(* CODESYS project SPT_Drives.library
   Company: Beckhoff Automation LLC
   DefaultNamespace: SPT_Drives
   Version: 3.0.2
   Placeholder: SPT Drives
   Title: SPT Drives

Project tree, tasks and I/O mapping:
  libraries: SPT Base Types, * (Beckhoff Automation LLC); SPT NC Axis, * (Beckhoff Automation LLC); Tc2_MC2, * (Beckhoff Automation GmbH); Tc2_NcDrive, * (Beckhoff Automation GmbH); Tc3_Module, * (Beckhoff Automation GmbH)
  Beckhoff/
    AX5000/
      function block FB_ResetRoutine_SoEDrive [ST]: Axis, CyclicLogic, Execute
    AX8000/
      function block FB_ResetRoutine_CoEDrive [ST]: Axis, CyclicLogic, Execute
  Project Information/
    function F_GetCompany [ST]
    function F_GetTitle [ST]
    function F_GetVersion [ST]
  Version/
    global variables Global_Version
*)

// Version/Global_Version
{attribute 'TcGenerated'}
{attribute 'no-analysis'}
{attribute 'linkalways'}
// This function has been automatically generated from the project information.
VAR_GLOBAL CONSTANT
	{attribute 'const_non_replaced'}
	stLibVersion_SPT_Drives : ST_LibVersion := (iMajor := 3, iMinor := 0, iBuild := 2, iRevision := 0, nFlags := 1, sVersion := '3.0.2');
END_VAR

// Beckhoff/AX5000/FB_ResetRoutine_SoEDrive
FUNCTION_BLOCK FINAL FB_ResetRoutine_SoEDrive EXTENDS FB_CyclicFB IMPLEMENTS I_MotionSequence
VAR_INPUT
END_VAR
VAR_OUTPUT
END_VAR
VAR
    _Axis : I_BasicAxis;
END_VAR

VAR
    MCReset      : MC_Reset;
    SoEReset     : FB_SoEReset;
    SequenceStep : UDINT;
END_VAR

PROPERTY Axis : I_BasicAxis
GET
Axis := _Axis;
END_GET
SET
_Axis := Axis;
END_SET
END_PROPERTY

METHOD PUBLIC  CyclicLogic
VAR_INPUT
END_VAR
CASE SequenceStep OF
    10:
        SoEReset(Axis := _Axis.Axis.NcToPlc, bExecute := TRUE);

        IF NOT SoEReset.bBusy THEN
            IF SoEReset.bError THEN
                _Error := TRUE;

                IF SoEReset.iSercosErrId < 0 THEN
                    _ErrorID := SoEReset.iSercosErrId;
                ELSE
                    _ErrorID := SoEReset.iAdsErrId;
                END_IF

                SequenceStep := 0;
            ELSE
                //No error occurred
                SequenceStep := SequenceStep + 10;
            END_IF

            SoEReset(Axis := _Axis.Axis.NcToPlc, bExecute := FALSE);
        END_IF

    20:
        MCReset(Axis := _Axis.Axis, Execute := TRUE);

        IF NOT MCReset.Busy THEN
            IF MCReset.Error THEN
                _Error   := TRUE;
                _ErrorID := MCReset.ErrorID;
            END_IF

            //Done
            SequenceStep := 0;
            MCReset(Axis := _Axis.Axis, Execute := FALSE);
        END_IF
END_CASE

_Busy := SequenceStep <> 0;
END_METHOD

METHOD PUBLIC Execute : BOOL
IF (_Axis = 0) OR _Busy THEN
    RETURN;
END_IF

_Busy        := TRUE;
_Error       := FALSE;
_ErrorID     := 0;
SequenceStep := 10;

Execute := TRUE;
END_METHOD

END_FUNCTION_BLOCK

// Beckhoff/AX8000/FB_ResetRoutine_CoEDrive
FUNCTION_BLOCK FINAL FB_ResetRoutine_CoEDrive EXTENDS FB_CyclicFB IMPLEMENTS I_MotionSequence
VAR_INPUT
END_VAR
VAR_OUTPUT
END_VAR
VAR
    _Axis : I_BasicAxis;
END_VAR

VAR
    MCReset : MC_Reset;
END_VAR

PROPERTY Axis : I_BasicAxis
GET
Axis := _Axis;
END_GET
SET
_Axis := Axis;
END_SET
END_PROPERTY

METHOD PUBLIC  CyclicLogic
VAR_INPUT
END_VAR
MCReset(Axis := _Axis.Axis, Busy => _Busy);

IF NOT MCReset.Busy THEN
    IF MCReset.Error THEN
        _Error   := TRUE;
        _ErrorID := MCReset.ErrorID;
    END_IF

    MCReset(Axis := _Axis.Axis, Execute := FALSE);
END_IF
END_METHOD

METHOD PUBLIC Execute : BOOL
IF (_Axis = 0) THEN
    RETURN;
END_IF

MCReset(Axis := _Axis.Axis, Execute := TRUE);

_Busy    := TRUE;
_Error   := FALSE;
_ErrorID := 0;

Execute := TRUE;
END_METHOD

END_FUNCTION_BLOCK

// Project Information/F_GetCompany
// This function has been automatically generated from the project information.
{attribute 'signature_flag' := '1073741824'}
{attribute 'TcGenerated'}
{attribute 'no-analysis'}
FUNCTION F_GetCompany : WSTRING
VAR_INPUT
	
END_VAR

F_GetCompany := "Beckhoff Automation LLC";

END_FUNCTION

// Project Information/F_GetTitle
// This function has been automatically generated from the project information.
{attribute 'signature_flag' := '1073741824'}
{attribute 'TcGenerated'}
{attribute 'no-analysis'}
FUNCTION F_GetTitle : WSTRING
VAR_INPUT
	
END_VAR

F_GetTitle := "SPT Drives";

END_FUNCTION

// Project Information/F_GetVersion
// This function has been automatically generated from the project information.
{attribute 'signature_flag' := '1073741824'}
{attribute 'TcGenerated'}
{attribute 'no-analysis'}
FUNCTION F_GetVersion : ST_LibVersion
VAR_INPUT
	
END_VAR

F_GetVersion.iMajor := 3;
F_GetVersion.iMinor := 0;
F_GetVersion.iBuild := 2;
F_GetVersion.iRevision := 0;
F_GetVersion.sVersion := '3.0.2';
F_GetVersion.nFlags := 1;

END_FUNCTION
